PROGRAM MAIN
VAR
END_VAR

END_PROGRAM

(* stored: Version 1.1.0.1
   POU MAIN: Id {36ebb702-e02f-4f1c-9425-8952b0cbb063} *)
